TYPE AX5000_P_0314 :
STRUCT
	Actual_lenght:UINT;
	Max_lenght:UINT;
	String_output_mode:UINT;
	Backlight_mode:UINT;
	Keypad_mode:UINT;
//	{attribute 'hide'}
	Rsvd:UINT;
	Output_string:STRING(39);
END_STRUCT
END_TYPE

(* stored: Version 1.1.0.1, ProductVersion 3.1.4024.4
   DUT AX5000_P_0314: Id {a8a7740c-f9a1-49d1-8a60-1dc4e76ccfd8} *)
